FUNCTION_BLOCK FB_RobotRegionMove_AllocatedConveyor EXTENDS FB_ObjectBase_V2 IMPLEMENTS IBasicElement
VAR_INPUT
    Robot     					: REFERENCE TO FB_FanucRobot_Basic;
	DifferenceCV 				: REFERENCE TO FB_motor;    // Allocated area feed in conveyor(diff and same size conveyor)
	SamesizeCV					: REFERENCE TO FB_motor;
//	SameSizeFullSensor 			: REFERENCE TO BOOL; 				 // Because the same size sensor implement FB_ConveyorSameSize, so use reference to connect it
   // Command   : ST_WareHouseWithRobotMove_Command;
   	cylinder : REFERENCE TO UNI_CylinderList;
   	Input : ST_InputTable;
    Info	  : ST_RobotRegionMove_Info;
	Stop	  : BOOL;
END_VAR
VAR_OUTPUT
  // Status : ST_WareHouseWithRobotMove_Status;
END_VAR
VAR
	_Abort		: BOOL;
	strStatus	: STRING;
	uiResumeStep : UINT;
	
	Area	: E_RobotArea :=E_RobotArea.TransmitCV;
	UseA 	: BOOL;
	UseB	: BOOL;
	SameSizeFullSensor 			: BOOL; 				 // Because the same size sensor implement FB_ConveyorSameSize, so use reference to connect it
	Get 	:BOOL;
	tonTimeOut	:TON;
	tonDelay	:TON;
	tonDelay_SameSizeGetBox : TON;
	tonDelay_SameSizeDelayBox : TON;
	tonFeedBoxTimeout : TON;
	_UniqueErrorCode :STRING;
	PreviousStrStatus : STRING;
	PreviousErrorCode : STRING;
END_VAR


SUPER^.A10_StateControl();
A00_BasicUnits();
SameSizeFullSensor := Input.bSameSizeCV_BoxNearStorageSensor;

ACTION A00_BasicUnits:
tonTimeOut(PT:=T#60S);
tonFeedBoxTimeout(PT:=T#30s);
tonDelay(PT:=T#1.5S);
tonDelay_SameSizeDelayBox(PT:=T#1.5S);
tonDelay_SameSizeGetBox(PT:=T#50MS);
ErrorID:=2210;
END_ACTION

METHOD M_CheckCommand : BOOL // True : Command is useful
VAR_INPUT
END_VAR
VAR
	
END_VAR
// Check command paremeter is correct
	
	THIS^.Get :=Info.Get;	
	UseA :=Info.UseA;
	UseB :=Info.UseB;
	
//Allocated/Empty conveyor
		IF UseA AND ( Info.A_Position<1 OR  Info.A_Position>2 ) THEN
			strStatus:='Wrong command ,Position A Not allow';
			M_CheckCommand:=FALSE;
			RETURN;		
		END_IF
	
		IF UseB AND ( Info.B_Position<1 OR  Info.B_Position>2 )THEN
			strStatus:='Wrong command ,Position B Not allow';
			M_CheckCommand:=FALSE;
			RETURN;		
		END_IF	
M_CheckCommand:=TRUE;
END_METHOD

METHOD M_CheckUnitsNotBusy : BOOL
VAR_INPUT
END_VAR
M_CheckUnitsNotBusy := true;
END_METHOD

METHOD M_CheckUnitsReady : BOOL
VAR_INPUT
END_VAR
M_CheckUnitsReady := true;
END_METHOD

METHOD  M_STATE_ABORTED
VAR_INPUT
END_VAR
ERROR :=TRUE;
Busy    := FALSE;
Aborted := TRUE;
Status := strStatus;
UniqueErrorCode:=_UniqueErrorCode;
_AbortCompleted:=FALSE;
IF NOT Execute THEN
	eSTATE:=STATE_RESETTING;
END_IF

IF Execute AND Reset THEN
	uiExecutingStep :=uiResumeStep;
	PreviousStrStatus := strStatus;
	PreviousErrorCode := _UniqueErrorCode;
	eSTATE:=STATE_EXECUTING;
END_IF
END_METHOD

METHOD  M_STATE_ABORTING
VAR_INPUT
END_VAR
CASE uiAbortingStep OF
	0 :
		uiAbortingStep:=9999;
		tonFeedBoxTimeout.IN :=FALSE;
		tonTimeOut.IN :=FALSE;
		tonDelay.IN :=FALSE;
		_Abort :=FALSE;
		DifferenceCV.M_MotorStop();
		SamesizeCV.M_MotorStop();
		IF strStatus = PreviousStrStatus THEN
			_UniqueErrorCode :=PreviousErrorCode;
		END_IF
		
	9999:	_AbortCompleted:=TRUE;
END_CASE

IF _AbortCompleted THEN	
	eSTATE :=STATE_ABORTED;
END_IF
END_METHOD

METHOD  M_STATE_DONE
VAR_INPUT
END_VAR
Busy := FALSE;
Done := TRUE;
IF NOT Execute THEN
    eState := STATE_RESETTING;
END_IF
END_METHOD

METHOD  M_STATE_DORMANT
VAR_INPUT
END_VAR
// Clear FB output
Busy            := FALSE;
Done            := FALSE;
Aborted         := FALSE;
Error           := FALSE;
ErrorID         := 0;
Status          := '';
_ResetCompleted := FALSE;
_Error          := FALSE;
_Executed       := FALSE;
tonDelay_SameSizeGetBox.IN := FALSE;
tonDelay_SameSizeDelayBox.IN :=false;
tonTimeOut.IN:=FALSE;
strStatus :='No Error';
uiExecutingStep :=uiResettingStep :=uiResumeStep :=0;
tonDelay.IN :=FALSE;
tonFeedBoxTimeout.IN :=FALSE;
_UniqueErrorCode :='0';
PreviousStrStatus			 :='';
PreviousErrorCode			 :='';
// Wait Execute command
IF Execute THEN
    eState := STATE_EXECUTING;
END_IF
END_METHOD

METHOD  M_STATE_ERROR
VAR_INPUT
END_VAR
ERROR   :=TRUE;
Busy	:=FALSE;
Status := strStatus;
UniqueErrorCode:=_UniqueErrorCode;
cylinder.List.fbSameSizeCV_Press3.M_Retract();
cylinder.List.fbSameSizeCV_Press4.M_Retract();
IF NOT Execute THEN	
eSTATE:=STATE_RESETTING;
END_IF
END_METHOD

METHOD  M_STATE_EXECUTING
VAR_INPUT
END_VAR
VAR_INST
	BoxReady_1st : BOOL;
	BoxReady_2nd : BOOL;
    uiBothStep : UINT;
    uiSingleClampStep : UINT;	
	Address_A : INT;
	Address_B : INT;
	bGetBoxInSameSizeConveyor : BOOL;
	uiSameGetBoxStep : UINT;
	bSameSizeCVMoveForward  : BOOL;
	bSameSizeCVMoveBackward : BOOL;
	bDiffCVMoveForward		:BOOL;
	bDiffCVMoveBackward		:BOOL;


END_VAR
VAR
	WareHouse: INT;
	
END_VAR
// Set Busy active edit by johnson
Busy := TRUE;
IF THIS^.Stop THEN // Pending the timeout when Stop signal occur
	tonTimeout.IN :=FALSE;
END_IF

IF bSameSizeCVMoveForward THEN
	IF NOT SamesizeCV.InBackWard THEN
		SamesizeCV.M_MoveForward();
	END_IF
END_IF
IF bSameSizeCVMoveBackward THEN
	IF NOT SamesizeCV.InForWard THEN
	 SamesizeCV.M_MoveBackward();
	END_IF
END_IF
IF bDiffCVMoveForward THEN
	IF NOT DifferenceCV.InBackWard THEN
		DifferenceCV.M_MoveForward();
	END_IF
END_IF
IF bDiffCVMoveBackward THEN
	IF NOT DifferenceCV.InForWard THEN
		DifferenceCV.M_MoveBackward();
	END_IF
END_IF


// Service Process
CASE uiExecutingStep OF
	0:
        // Clear variable
        uiBothStep := 0;
		uiSingleClampStep :=0;
		BoxReady_1st := 0;
		BoxReady_2nd := 0;
		tonTimeOut.IN:=FALSE;
		bSameSizeCVMoveForward  :=FALSE;
		bSameSizeCVMoveBackward :=FALSE;
		bDiffCVMoveForward		:=FALSE;
		bDiffCVMoveBackward		:=FALSE;
        // Check command
        IF M_CheckCommand() THEN
            uiExecutingStep := 10;
		ELSE
			_Error:=TRUE;
        END_IF
    10:
        // Start process, check units first
        IF M_CheckUnitsReady() THEN
            uiExecutingStep := 20;
        END_IF
    20:
        // CHeck units not busy state
        IF M_CheckUnitsNotBusy() THEN
            uiExecutingStep := 1000;
        END_IF
   
	1000:   
			// Read   coordinate
			 Area := THIS^.Area;
 			 Address_A := LREAL_TO_INT(Info.A_Position);
			 Address_B := LREAL_TO_INT(Info.B_Position);
			 bGetBoxInSameSizeConveyor := Get AND ((UseA AND Address_A=2) OR (UseB AND Address_B=2));
			 IF bGetBoxInSameSizeConveyor THEN
				 cylinder.List.fbSameSizeCV_Press3.M_Retract();
				 cylinder.List.fbSameSizeCV_Press4.M_Retract();
			 END_IF
			 uiSameGetBoxStep :=0;
			 tonDelay_SameSizeGetBox.IN:=FALSE;
			IF UseA AND NOT UseB THEN
				//Only clampA
				uiExecutingStep := 10000;
			ELSIF NOT UseA AND UseB THEN
				//Only ClampB 
				uiExecutingStep := 20000;
			ELSIF UseA AND UseB THEN
				//Both Clamps
				uiExecutingStep := 30000;		
			END_IF
       
    10000: // Only ClampA 
        IF NOT Robot._DI1.Done THEN
            
            
			CASE uiSingleClampStep OF
				
				0://
					 IF Get THEN // Get box job
//						IF FeedInConveyor.P_PermitCommand AND NOT FeedInConveyor.P_isRunningBackward THEN
//            				FeedInConveyor.M_AutoMoveReverse(sRecordSource := '');
//						END_IF
//						IF 
					 	
						CASE Address_A OF
							1:
								tonDelay.IN :=Input.bDifferentSizeCV_BoxDetect7_Sensor;
								bDiffCVMoveBackward:=TRUE;
								bDiffCVMoveForward:=FALSE;
								DifferenceCV.M_MoveBackward();
								
							2:
								CASE uiSameGetBoxStep OF
									0:
									//tonDelay.IN :=SameSizeFullSensor;	
									bSameSizeCVMoveBackward := TRUE;
									bSameSizeCVMoveForward := FALSE;
									SamesizeCV.M_MoveBackward();
									cylinder.List.fbSameSizeCV_Press3.M_Retract();
									cylinder.List.fbSameSizeCV_Press4.M_Retract();
									uiSameGetBoxStep :=100;
									
									100:
										tonDelay_SameSizeGetBox.IN := Input.bSameSizeCV_BoxDetect6_Sensor;
										IF tonDelay_SameSizeGetBox.Q THEN
											cylinder.List.fbSameSizeCV_Press3.M_Extend();
											uiSameGetBoxStep :=200;
										END_IF
									200:
										tonDelay_SameSizeGetBox.IN:=FALSE;
										tonDelay_SameSizeDelayBox.IN :=SameSizeFullSensor;
										IF 	tonDelay_SameSizeDelayBox.Q THEN
											uiSameGetBoxStep :=300;
										END_IF	
									300:
										cylinder.List.fbSameSizeCV_Press4.M_Extend();
										tonDelay.IN :=TRUE;
										uiSameGetBoxStep :=400;
									400: 
										IF tonDelay.Q THEN
											cylinder.List.fbSameSizeCV_Press4.M_Retract();
										END_IF
								END_CASE
						END_CASE	
			
					ELSE
//						IF FeedInConveyor.P_PermitCommand AND NOT FeedInConveyor.P_isRunningBackward THEN
//            				FeedInConveyor.M_MoveForward(sRecordSource := '');
//						END_IF
						CASE Address_A OF
							1:
								tonDelay.IN := NOT Input.bDifferentSizeCV_BoxDetect7_Sensor;
								bDiffCVMoveForward :=TRUE;
								bDiffCVMoveBackward:=FALSE;
								DifferenceCV.M_MoveForward();
							2:
								tonDelay.IN :=NOT SameSizeFullSensor;
								bSameSizeCVMoveForward :=TRUE;
								bSameSizeCVMoveBackward:=FALSE;
								SamesizeCV.M_MoveForward();			
						END_CASE					
				
					END_IF	
				
						IF tonDelay.Q THEN
							tonFeedBoxTimeout.IN :=FALSE;
							uiSingleClampStep:=1000;
						END_IF
						tonFeedBoxTimeout.IN :=TRUE;
						IF tonFeedBoxTimeout.Q THEN
							tonFeedBoxTimeout.IN :=FALSE;
							strStatus :='Feed Box timeout';
							uiResumeStep:=10000;
							_Abort:=TRUE;
						END_IF
				1000:
						BoxReady_1st:=TRUE;
						tonDelay.IN:=FALSE;
						bSameSizeCVMoveForward  :=FALSE;
						bSameSizeCVMoveBackward :=FALSE;
						bDiffCVMoveForward		:=FALSE;
						bDiffCVMoveBackward		:=FALSE;						
						DifferenceCV.M_MotorStop();
						SamesizeCV.M_MotorStop();
						uiSingleClampStep:=9999;
				9999: //Wait	
			END_CASE
			          		 
				  // Robot Abs move
           		 Robot.M_StartRobotAbsMove(GetBox:=Get,
											UseClampA:=UseA,
											UseClampB:=UseB,
											Area:=Area,
											ClampA_Address:=Address_A,
											ClampB_Address:=Address_B,
											BoxReady_1:=BoxReady_1st,
											BoxReady_2:=BoxReady_2nd);				  
		
        ELSE
			tonTimeOut.IN:=FALSE;
            uiExecutingStep := 10080;
        END_IF
		tonTimeOut.IN:=TRUE;
		IF tonTimeOut.Q=TRUE THEN
			tonTimeOut.IN:=FALSE;
			strStatus :='Robot move timeout';
			_Error:=TRUE;
		END_IF	
    10080:
        Robot.M_ResetRobotAbsMove(UseA,UseB); // Clear command and go to place box
		tonTimeOut.IN:=TRUE;
		uiSameGetBoxStep:=0;
        IF NOT Robot._DI1.Done THEN
			tonTimeOut.IN:=FALSE;
            uiExecutingStep := 50000; 
        END_IF
		
    	IF tonTimeOut.Q=TRUE THEN
			strStatus :='Reset Robot timeout';
			_Error:=TRUE;
		END_IF	
    
   20000: // Only ClampB
        IF NOT Robot._DI1.Done THEN
            			
			CASE uiSingleClampStep OF
			0:	
					 IF Get THEN // Get box job
//						IF FeedInConveyor.P_PermitCommand AND NOT FeedInConveyor.P_isRunningBackward THEN
//            				FeedInConveyor.M_AutoMoveReverse(sRecordSource := '');
//						END_IF
//						IF 
					 	
						CASE Address_B OF
							1:
								tonDelay.IN :=Input.bDifferentSizeCV_BoxDetect7_Sensor;
								bDiffCVMoveBackward:=TRUE;
								bDiffCVMoveForward := FALSE;
								DifferenceCV.M_MoveBackward();
								
							2:
//								tonDelay.IN :=SameSizeFullSensor;	
//								SamesizeCV.M_MoveBackward();
//								cylinder.List.fbSameSizeCV_Press3.M_Retract();
//								cylinder.List.fbSameSizeCV_Press4.M_Retract();
								CASE uiSameGetBoxStep OF
									0:
									//tonDelay.IN :=SameSizeFullSensor;	
									bSameSizeCVMoveForward :=FALSE;
									bSameSizeCVMoveBackward := TRUE;
									SamesizeCV.M_MoveBackward();
									cylinder.List.fbSameSizeCV_Press3.M_Retract();
									cylinder.List.fbSameSizeCV_Press4.M_Retract();
									uiSameGetBoxStep :=100;
									
									100:
										tonDelay_SameSizeGetBox.IN := Input.bSameSizeCV_BoxDetect6_Sensor;
										IF tonDelay_SameSizeGetBox.Q THEN
											cylinder.List.fbSameSizeCV_Press3.M_Extend();
											uiSameGetBoxStep :=200;
										END_IF
									200:
										tonDelay_SameSizeGetBox.IN:=FALSE;
										tonDelay_SameSizeDelayBox.IN :=SameSizeFullSensor;
										IF 	tonDelay_SameSizeDelayBox.Q THEN
											uiSameGetBoxStep :=300;
										END_IF	
									300:
										cylinder.List.fbSameSizeCV_Press4.M_Extend();
										uiSameGetBoxStep :=400;
									400: 
										tonDelay.IN :=TRUE;
										IF tonDelay.Q THEN
											cylinder.List.fbSameSizeCV_Press4.M_Retract();
										END_IF
								END_CASE			

						END_CASE	
			
					ELSE
//						IF FeedInConveyor.P_PermitCommand AND NOT FeedInConveyor.P_isRunningBackward THEN
//            				FeedInConveyor.M_MoveForward(sRecordSource := '');
//						END_IF
						CASE Address_B OF
							1:
								tonDelay.IN := NOT Input.bDifferentSizeCV_BoxDetect7_Sensor;
								bDiffCVMoveForward	:=TRUE;
								bDiffCVMoveBackward	:=FALSE;
								DifferenceCV.M_MoveForward();
							2:
								tonDelay.IN :=NOT SameSizeFullSensor;
								bSameSizeCVMoveForward :=TRUE;
								bSameSizeCVMoveBackward :=FALSE;
								SamesizeCV.M_MoveForward();			
						END_CASE					
				
					END_IF	
				
						IF tonDelay.Q THEN
							tonFeedBoxTimeout.IN :=FALSE;
							uiSingleClampStep:=1000;
						END_IF
						tonFeedBoxTimeout.IN :=TRUE;
						IF tonFeedBoxTimeout.Q THEN
							tonFeedBoxTimeout.IN :=FALSE;
							strStatus :='Feed Box timeout';
							uiResumeStep:=10000;
							_Abort:=TRUE;
						END_IF
				1000:
						//BoxReady_1st:=TRUE;
						BoxReady_2nd:=TRUE;
						tonDelay.IN:=FALSE;
						bSameSizeCVMoveForward  :=FALSE;
						bSameSizeCVMoveBackward :=FALSE;
						bDiffCVMoveForward		:=FALSE;
						bDiffCVMoveBackward		:=FALSE;
						DifferenceCV.M_MotorStop();
						SamesizeCV.M_MotorStop();
						uiSingleClampStep:=9999;
				9999: //Wait	

			END_CASE
			          		 
				  // Robot Abs move
           		 Robot.M_StartRobotAbsMove( GetBox:=Get,
											UseClampA:=UseA,
											UseClampB:=UseB,
											Area:=Area,
											ClampA_Address:=Address_A,
											ClampB_Address:=Address_B,
											BoxReady_1:=BoxReady_1st,
											BoxReady_2:=BoxReady_2nd);	
        ELSE
			tonTimeOut.IN:=FALSE;
            uiExecutingStep := 20080;
        END_IF
		tonTimeOut.IN:=TRUE;
		IF tonTimeOut.Q=TRUE THEN
			tonTimeOut.IN:=FALSE;
			strStatus :='Robot move timeout';
			_Error:=TRUE;
		END_IF	
    20080:
       Robot.M_ResetRobotAbsMove(UseA,UseB);; // Clear command 
		uiSameGetBoxStep :=0;
        IF NOT Robot._DI1.Done THEN
            uiExecutingStep := 50000; 
        END_IF
		tonTimeOut.IN:=TRUE;
		IF tonTimeOut.Q=TRUE THEN
			strStatus :='Reset Robot timeout';
			_Error:=TRUE;
		END_IF	
    30000: // Both Clamps
        		
		
		  CASE uiBothStep OF
           		0://	
					BoxReady_1st := FALSE;
					BoxReady_2nd := FALSE;					
					uiBothStep:=1000;						
				
				1000:
						IF Get THEN // Get box job
							CASE Address_A OF
								1:
									tonDelay.IN :=Input.bDifferentSizeCV_BoxDetect7_Sensor;
									bDiffCVMoveForward	:=FALSE;
									bDiffCVMoveBackward	:=TRUE;
									DifferenceCV.M_MoveBackward();
									
								2:
//									tonDelay.IN :=SameSizeFullSensor;	
//									SamesizeCV.M_MoveBackward();
//									cylinder.List.fbSameSizeCV_Press3.M_Retract();
//									cylinder.List.fbSameSizeCV_Press4.M_Retract();
								CASE uiSameGetBoxStep OF
									0:
									//tonDelay.IN :=SameSizeFullSensor;	
									bSameSizeCVMoveForward  :=FALSE;
									bSameSizeCVMoveBackward :=TRUE;
									SamesizeCV.M_MoveBackward();
									cylinder.List.fbSameSizeCV_Press3.M_Retract();
									cylinder.List.fbSameSizeCV_Press4.M_Retract();
									uiSameGetBoxStep :=100;
									
									100:
										tonDelay_SameSizeGetBox.IN := Input.bSameSizeCV_BoxDetect6_Sensor;
										IF tonDelay_SameSizeGetBox.Q THEN
											cylinder.List.fbSameSizeCV_Press3.M_Extend();
											uiSameGetBoxStep :=200;
										END_IF
									200:
										tonDelay_SameSizeGetBox.IN:=FALSE;
										tonDelay_SameSizeDelayBox.IN :=SameSizeFullSensor;
										IF 	tonDelay_SameSizeDelayBox.Q THEN
											uiSameGetBoxStep :=300;
										END_IF	
									300:
										cylinder.List.fbSameSizeCV_Press4.M_Extend();
										tonDelay.IN :=TRUE;
										uiSameGetBoxStep :=400;
									400: 
										IF tonDelay.Q THEN
											cylinder.List.fbSameSizeCV_Press4.M_Retract();
										END_IF
								END_CASE
				
							END_CASE	
			
						ELSE
							CASE Address_A OF
								1:
									tonDelay.IN := NOT Input.bDifferentSizeCV_BoxDetect7_Sensor;
									bDiffCVMoveForward	:=TRUE;
									bDiffCVMoveBackward	:=FALSE;
									DifferenceCV.M_MoveForward();
								2:
									tonDelay.IN :=NOT SameSizeFullSensor;
									bSameSizeCVMoveForward  :=TRUE;
									bSameSizeCVMoveBackward :=FALSE;
									SamesizeCV.M_MoveForward();			
							END_CASE					
				
						END_IF	
				
						IF tonDelay.Q THEN
							tonFeedBoxTimeout.IN :=FALSE;
							uiSameGetBoxStep:=0;
							uiBothStep:=2000;
						END_IF
						tonFeedBoxTimeout.IN :=TRUE;
						IF tonFeedBoxTimeout.Q THEN
							tonFeedBoxTimeout.IN :=FALSE;
							strStatus :='Feed Box timeout';
							uiResumeStep:=30000;
							_Abort:=TRUE;
						END_IF
				2000:
						tonDelay.IN :=FALSE;
						bSameSizeCVMoveForward  :=FALSE;
						bSameSizeCVMoveBackward :=FALSE;
						bDiffCVMoveForward		:=FALSE;
						bDiffCVMoveBackward		:=FALSE;
						DifferenceCV.M_MotorStop();
						SamesizeCV.M_MotorStop();
						BoxReady_1st:=TRUE;
						tonDelay_SameSizeGetBox.IN := FALSE;
						tonDelay_SameSizeDelayBox.IN :=FALSE;
						IF Robot._DI1.Notification THEN
							uiBothStep:=3000;
						END_IF
				3000:
						IF Get THEN // Get box job
							CASE Address_B OF
								1:
									tonDelay.IN :=Input.bDifferentSizeCV_BoxDetect7_Sensor;
									bDiffCVMoveForward	:=FALSE;
									bDiffCVMoveBackward :=TRUE;
									DifferenceCV.M_MoveBackward();
									
								2:
//									tonDelay.IN :=SameSizeFullSensor;	
//									SamesizeCV.M_MoveBackward();
//									cylinder.List.fbSameSizeCV_Press3.M_Retract();
//									cylinder.List.fbSameSizeCV_Press4.M_Retract();
									CASE uiSameGetBoxStep OF
									0:
									//tonDelay.IN :=SameSizeFullSensor;	
									bSameSizeCVMoveForward :=FALSE;
									bSameSizeCVMoveBackward :=TRUE;
									SamesizeCV.M_MoveBackward();
									cylinder.List.fbSameSizeCV_Press3.M_Retract();
									cylinder.List.fbSameSizeCV_Press4.M_Retract();
									uiSameGetBoxStep :=100;
									
									100:
										tonDelay_SameSizeGetBox.IN := Input.bSameSizeCV_BoxDetect6_Sensor;
										IF tonDelay_SameSizeGetBox.Q THEN
											cylinder.List.fbSameSizeCV_Press3.M_Extend();
											uiSameGetBoxStep :=200;
										END_IF
									200:
										tonDelay_SameSizeGetBox.IN:=FALSE;
										tonDelay_SameSizeDelayBox.IN :=SameSizeFullSensor;
										IF 	tonDelay_SameSizeDelayBox.Q THEN
											uiSameGetBoxStep :=300;
										END_IF	
									300:
										cylinder.List.fbSameSizeCV_Press4.M_Extend();
										tonDelay.IN :=TRUE;
										uiSameGetBoxStep :=400;
									400: 
										IF tonDelay.Q THEN
											cylinder.List.fbSameSizeCV_Press4.M_Retract();
										END_IF
								END_CASE
							END_CASE	
			
						ELSE
							CASE Address_B OF
								1:
									tonDelay.IN := NOT Input.bDifferentSizeCV_BoxDetect7_Sensor;
									bDiffCVMoveForward	:=TRUE;
									bDiffCVMoveBackward := FALSE;
									DifferenceCV.M_MoveForward();
								2:
									tonDelay.IN :=NOT SameSizeFullSensor;
									bSameSizeCVMoveForward :=TRUE;
									bSameSizeCVMoveBackward := FALSE;
									SamesizeCV.M_MoveForward();			
							END_CASE					
				
						END_IF	
				
						IF tonDelay.Q THEN
							tonFeedBoxTimeout.IN :=FALSE;
							uiBothStep:=9000;
						END_IF
						IF tonFeedBoxTimeout.Q THEN
							tonFeedBoxTimeout.IN :=FALSE;
							strStatus :='Feed Box timeout';
							uiResumeStep:=30000;
							_Abort:=TRUE;
						END_IF
				
				9000:
						BoxReady_2nd:=TRUE;
						tonDelay.IN :=FALSE;
						bSameSizeCVMoveForward  :=FALSE;
						bSameSizeCVMoveBackward :=FALSE;
						bDiffCVMoveForward		:=FALSE;
						bDiffCVMoveBackward		:=FALSE;
						DifferenceCV.M_MotorStop();
						SamesizeCV.M_MotorStop();
				
					
       
      	  END_CASE

       	  // Robot Abs move
           		 Robot.M_StartRobotAbsMove( GetBox:=Get,
											UseClampA:=UseA,
											UseClampB:=UseB,
											Area:=Area,
											ClampA_Address:=Address_A,
											ClampB_Address:=Address_B,
											BoxReady_1:=BoxReady_1st,
											BoxReady_2:=BoxReady_2nd);	
		
		
        IF Robot._DI1.Done THEN
			tonTimeOut.IN:=FALSE;
            uiExecutingStep := 30080;
        END_IF
			tonTimeOut.IN:=TRUE;
		IF tonTimeOut.Q=TRUE THEN
			tonTimeOut.IN:=FALSE;
			strStatus :='Robot move timeout';
			_Abort:=TRUE;
		END_IF
    30080: // Check robot command is clear
        
        Robot.M_ResetRobotAbsMove(UseA,UseB);

        IF NOT Robot._DI1.Done THEN
			tonTimeOut.IN:=FALSE;
            uiExecutingStep := 50000; // go to place step
        END_IF    
   		tonTimeOut.IN:=TRUE;
		IF tonTimeOut.Q=TRUE THEN
			strStatus :='Stop Robot timeout';
			_Error:=TRUE;
		END_IF	
  	50000:	// if robot put need box forward more time
			IF NOT Get THEN
				uiExecutingStep :=51000;
			ELSE
				uiExecutingStep :=99000;
			END_IF
    51000:	//conveyor forward 
			IF UseA THEN
				CASE Address_A OF
					1:
						tonDelay.IN := NOT Input.bDifferentSizeCV_BoxDetect7_Sensor;
						DifferenceCV.M_MoveForward();
					2:
						tonDelay.IN :=NOT SameSizeFullSensor;
						SamesizeCV.M_MoveForward();			
				END_CASE
			END_IF					
			IF UseB THEN
				CASE Address_B OF
					1:
						tonDelay.IN := NOT Input.bDifferentSizeCV_BoxDetect7_Sensor;
						DifferenceCV.M_MoveForward();
					2:
						tonDelay.IN :=NOT SameSizeFullSensor;
						SamesizeCV.M_MoveForward();			
				END_CASE
			END_IF
						IF tonDelay.Q THEN
							tonFeedBoxTimeout.IN :=FALSE;
							uiExecutingStep:=99000;
						END_IF
						IF tonFeedBoxTimeout.Q THEN
							tonFeedBoxTimeout.IN :=FALSE;
							strStatus :='Feed Box timeout';
							uiResumeStep:=30000;
							_Abort:=TRUE;
						END_IF
    99000: // process done
         Status    := 'Process completed';
		 bSameSizeCVMoveForward  :=FALSE;
		 bSameSizeCVMoveBackward :=FALSE;
		 bDiffCVMoveForward		:=FALSE;
		 bDiffCVMoveBackward		:=FALSE;
		 cylinder.List.fbSameSizeCV_Press3.M_Retract();
		 cylinder.List.fbSameSizeCV_Press4.M_Retract();
        _Executed := TRUE;
END_CASE
IF _Executed THEN
    eState := STATE_DONE;
ELSIF _Error THEN
	//FUN_UniqueErrorCodeGenerator(iErrorID := ErrorID,UinqueErrorCode=>_UniqueErrorCode);
	eState := STATE_ERROR;
ELSIF NOT Execute THEN
    eState := STATE_RESETTING;
END_IF
IF _Abort OR Abort THEN
	//FUN_UniqueErrorCodeGenerator(iErrorID := ErrorID,UinqueErrorCode=>_UniqueErrorCode);
	eSTATE:=STATE_ABORTING;
END_IF
END_METHOD

METHOD  M_STATE_RESETTING
VAR_INPUT
END_VAR
Error :=FALSE;
Done :=FALSE;
Busy := FALSE;


CASE uiResettingStep OF
	
	0:
		tonTimeOut.IN:=FALSE;
		tonDelay_SameSizeDelayBox.IN :=FALSE;
		Robot.M_ResetAllCommand();
		Robot.M_ResetRobotAbsMove(TRUE,TRUE);
		DifferenceCV.M_MotorStop();
		SamesizeCV.M_MotorStop();
		cylinder.List.fbSameSizeCV_Press3.M_Retract();
		cylinder.List.fbSameSizeCV_Press4.M_Retract();
		uiResettingStep:=100;
		
	100:	
	
		uiResettingStep:=9999;
	9999:
		_ResetCompleted:=TRUE;
END_CASE
IF _ResetCompleted THEN
	eSTATE:=STATE_DORMANT;
END_IF
END_METHOD

END_FUNCTION_BLOCK

(* stored: Version 1.1.0.1, ProductVersion 3.1.4024.13
   POU FB_RobotRegionMove_AllocatedConveyor: Id {b872a835-1d75-4fdc-8270-a8c157b9bdf9}, SpecialFunc None
   Folder Method: Id {a4239636-7ee3-4895-a57f-25269708e78a}
   Folder State: Id {7a280747-8a3a-44cf-81bf-eeed27a38ec8}
   Action A00_BasicUnits: Id {8689e687-336d-4ea9-8d03-cc4be06e76ed}
   Method M_CheckCommand: Id {a0a56b2c-4a8e-4c84-9511-f934763f5581}
   Method M_CheckUnitsNotBusy: Id {bd699f8a-95b7-4794-a4f8-0f5a8d076bda}
   Method M_CheckUnitsReady: Id {c157d73f-43b9-43cf-b386-ee2652830f33}
   Method M_STATE_ABORTED: Id {545087cf-44b0-4b0c-9d9c-06ac12763b96}
   Method M_STATE_ABORTING: Id {272367ac-711e-4377-9234-10bb14ffed4a}
   Method M_STATE_DONE: Id {995b98d7-79de-40b8-b4db-bcd57e12d7cd}
   Method M_STATE_DORMANT: Id {54c771d1-5869-4b0f-b1c8-039798218fc6}
   Method M_STATE_ERROR: Id {ca523e99-edc6-46b6-9c52-ae0823ef3080}
   Method M_STATE_EXECUTING: Id {074a31ee-2180-4eb9-8692-a35ade6092c7}
   Method M_STATE_RESETTING: Id {f1009dde-1906-4ace-a6ac-b1d2a7de8631} *)
